PROGRAM MAIN
VAR
END_VAR

SMTP();
SMTPFull();

END_PROGRAM

(* stored: Version 1.1.0.1, ProductVersion 3.1.4026.18
   POU MAIN: Id {5726de7a-92b0-4d31-a45f-7d6601e9be82}, SpecialFunc None *)
